RoboDK station: 01B - Inspection.rdk

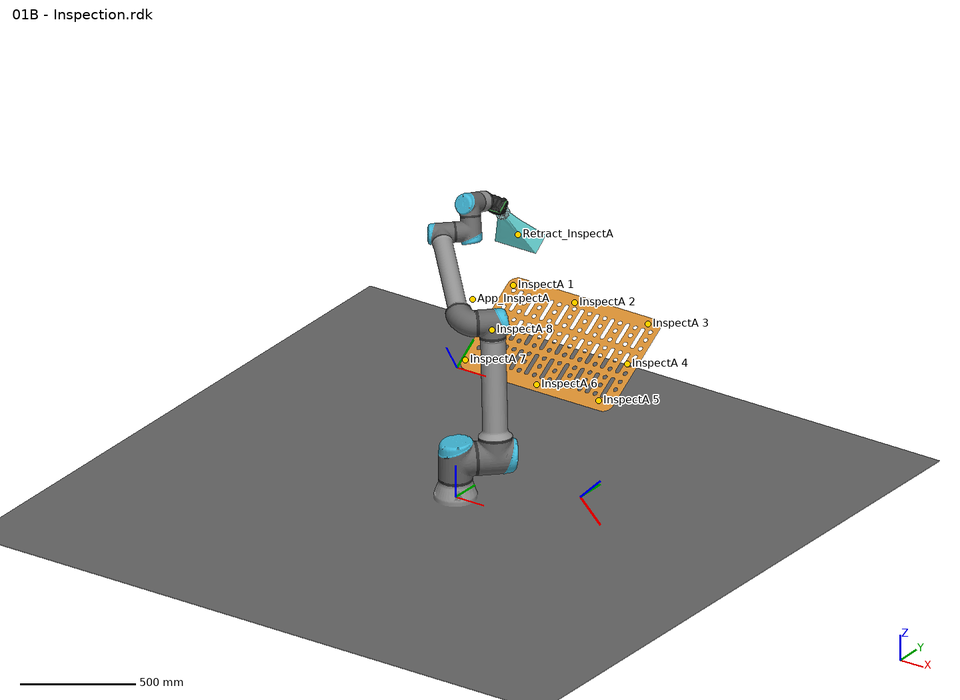
[picture v0: the station drawn from its stored meshes, robots at their saved joint values, targets as dots, program paths as lines]
Station 01B - Inspection (saved by RoboDK 5.4.1). Poses are relative to the parent item; angles as X-Y-Z fixed-axis rotations.
Station parameters (name, value as stored): Palletizing Plugin, LIN64
  - frame UR10e Base at (0, 0, 0) mm
    - robot UR10e: 6 axes, payload 10 kg, reach 1300 mm, repeatability 0.05 mm, weight 28.9 kg
        modified DH rows (alpha deg, a mm, theta deg, d mm): 0, 0, 0, 180.7; 90, 0, 180, 0; 0, 612.6, 0, 0; 0, 571.335, 0, 174.15; -90, 0, 0, 119.85; 90, 0, 180, 116.55
        joint limits [-360, -360, -360, -360, -360, -360] to [360, 360, 360, 360, 360, 360]; home [0, -90, -90, 0, 90, 0]; saved at [134.554, -97.678, -64.208, -41.542, 47.905, 196.197]
      - tool Camera 2, TCP at (0, -175.95, 321.06) mm, rotated rx 40 ry 0 rz 0 deg, size 215.7 x 276.1 x 372.4 mm
  - frame Frame Inspection A at (-380.72, 555.26, 295.21) mm, rotated rx 32.84 ry 0 rz 0 deg
    - object Inspection A at (0, 0, 0) mm, size 800 x 500 x 0 mm, geometry from Inspection A.step
  - frame Frame Inspection B at (727.24, -100, 245.26) mm, rotated rx 0 ry 45.31 rz 0 deg
    - object Inspection B at (0, 0, 0) mm, size 202.5 x 1023.2 x 500 mm, geometry from Inspection B.step
  - frame World at (0, 0, 0) mm
    - object Floor at (0, 0, -7) mm, size 3000 x 3000 x 4.2 mm, geometry from Floor.step
    - target InspectA 1 (Cartesian target) at (-347.72, 934.1, 545.69) mm, rotated rx 147.16 ry 0 rz 180 deg; joints [136.641, -92.365, -93.579, -18.27, 45.996, 197.35] of UR10e
    - target InspectA 2 (Cartesian target) at (-29.4, 940.44, 549.78) mm, rotated rx 147.16 ry 0 rz 180 deg; joints [110.562, -84.565, -101.198, -12.489, 70.392, 186.315] of UR10e
    - target InspectA 3 (Cartesian target) at (354.45, 944.76, 552.57) mm, rotated rx 147.16 ry 0 rz 180 deg; joints [73.379, -94.715, -90.86, -12.285, 105.862, 174.967] of UR10e
    - target InspectA 4 (Cartesian target) at (368.7, 765.58, 436.91) mm, rotated rx 147.16 ry 0 rz 180 deg; joints [65.973, -83.5, -113.681, -1.498, 112.895, 172.508] of UR10e
    - target InspectA 5 (Cartesian target) at (341.95, 589.35, 323.16) mm, rotated rx 147.16 ry 0 rz 180 deg; joints [58.371, -72.792, -134.071, 6.931, 120.071, 169.701] of UR10e
    - target InspectA 6 (Cartesian target) at (24.03, 579.19, 316.6) mm, rotated rx 147.16 ry 0 rz 180 deg; joints [137.912, -36.028, -147.589, -21.116, 44.84, 198.089] of UR10e
    - target InspectA 7 (Cartesian target) at (-359.2, 588.87, 322.85) mm, rotated rx 147.16 ry 0 rz 180 deg; joints [172.544, -63.266, -132.389, -51.549, 18.664, 246.078] of UR10e
    - target InspectA 8 (Cartesian target) at (-322.55, 735.63, 417.58) mm, rotated rx 147.16 ry 0 rz 180 deg; joints [151.927, -75.225, -120.876, -17.169, 32.534, 208.949] of UR10e
    - target App_InspectA (Cartesian target) at (-347.72, 629.23, 601.32) mm, rotated rx 147.16 ry 0 rz 180 deg; joints [166.44, -64.901, -105.974, -61.914, 21.743, 230.733] of UR10e
    - target Retract_InspectA (Cartesian target) at (-347.72, 967.63, 778.19) mm, rotated rx 147.16 ry 0 rz 180 deg; joints [134.554, -97.678, -64.208, -41.542, 47.905, 196.197] of UR10e
  - Python program main1-2 (listed below)

--- Python program main1-2 ---
from robodk.robolink import *      # RoboDK's API
from robodk.robomath import *      # Math toolbox for robots

RL = Robolink()

robot = RL.Item('UR10e')

app_InspectA = RL.Item('App_InspectA')
retract_InspectA = RL.Item('Retract_InspectA')

def moveRobot():
    robot.MoveL(app_InspectA)
    moveTargets(8)
    robot.MoveL(retract_InspectA)

def moveTargets(targets):
    for i in range(1, targets):
        targetName = f"InspectA {i}"
        robot.MoveJ(RL.Item(targetName))

moveRobot()
